ABB RAPID module: PersistentVars.mod

MODULE PersistentVars(SYSMODULE)
    PERS jointtarget calib_jointtargets{calib_array_size};
    PERS robtarget calib_robtargets{calib_array_size};
ENDMODULE
